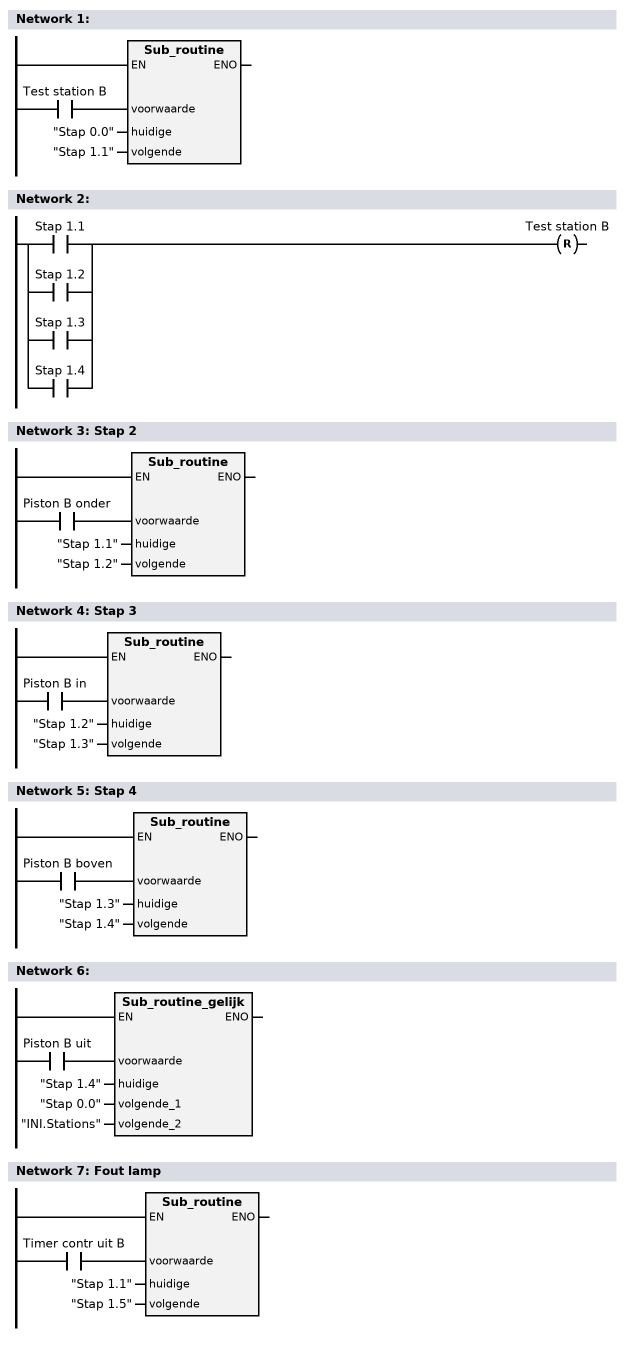
NETWORK
TITLE =
      A     "Test station B";
      =     L 0.0;
      BLD   103;
      CALL  "Sub_routine" (
           voorwaarde               := L 0.0,
           huidige                  := "Stap 0.0",
           volgende                 := "Stap 1.1");
      NOP   0;
NETWORK
TITLE =
      O     "Stap 1.1";
      O     "Stap 1.2";
      O     "Stap 1.3";
      O     "Stap 1.4";
      R     "Test station B";
NETWORK
TITLE = Stap 2
      A     "Piston B onder";
      =     L 0.0;
      BLD   103;
      CALL  "Sub_routine" (
           voorwaarde               := L 0.0,
           huidige                  := "Stap 1.1",
           volgende                 := "Stap 1.2");
      NOP   0;
NETWORK
TITLE = Stap 3
      A     "Piston B in";
      =     L 0.0;
      BLD   103;
      CALL  "Sub_routine" (
           voorwaarde               := L 0.0,
           huidige                  := "Stap 1.2",
           volgende                 := "Stap 1.3");
      NOP   0;
NETWORK
TITLE = Stap 4
      A     "Piston B boven";
      =     L 0.0;
      BLD   103;
      CALL  "Sub_routine" (
           voorwaarde               := L 0.0,
           huidige                  := "Stap 1.3",
           volgende                 := "Stap 1.4");
      NOP   0;
NETWORK
TITLE =
      A     "Piston B uit";
      =     L 0.0;
      BLD   103;
      CALL  "Sub_routine_gelijk" (
           voorwaarde               := L 0.0,
           huidige                  := "Stap 1.4",
           volgende_1               := "Stap 0.0",
           volgende_2               := "INI.Stations");
      NOP   0;
NETWORK
TITLE = Fout lamp
      A     "Timer contr uit B";
      =     L 0.0;
      BLD   103;
      CALL  "Sub_routine" (
           voorwaarde               := L 0.0,
           huidige                  := "Stap 1.1",
           volgende                 := "Stap 1.5");
      NOP   0;
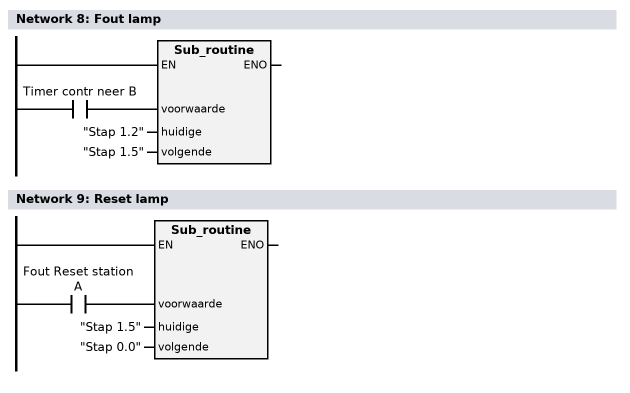
NETWORK
TITLE = Fout lamp
      A     "Timer contr neer B";
      =     L 0.0;
      BLD   103;
      CALL  "Sub_routine" (
           voorwaarde               := L 0.0,
           huidige                  := "Stap 1.2",
           volgende                 := "Stap 1.5");
      NOP   0;
NETWORK
TITLE = Reset lamp
      A     "Fout Reset station A";
      =     L 0.0;
      BLD   103;
      CALL  "Sub_routine" (
           voorwaarde               := L 0.0,
           huidige                  := "Stap 1.5",
           volgende                 := "Stap 0.0");
      NOP   0;
END_FUNCTION

FUNCTION "Simulatie_Run" : VOID	// FC 5
VERSION : 0.1
BEGIN
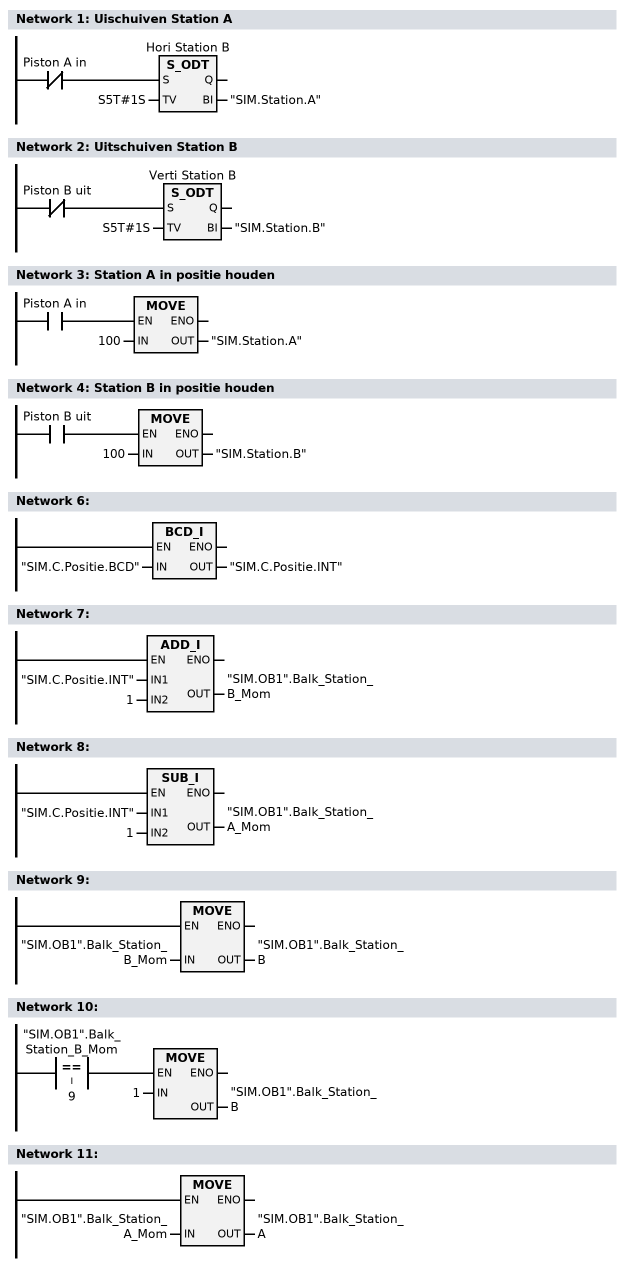
NETWORK
TITLE = Uischuiven Station A
      AN    "Piston A in";
      L     S5T#1S;
      SD    "Hori Station B";
      NOP   0;
      L     "Hori Station B";
      T     "SIM.Station.A";
      NOP   0;
      NOP   0;
NETWORK
TITLE = Uitschuiven Station B
      AN    "Piston B uit";
      L     S5T#1S;
      SD    "Verti Station B";
      NOP   0;
      L     "Verti Station B";
      T     "SIM.Station.B";
      NOP   0;
      NOP   0;
NETWORK
TITLE = Station A in positie houden
      A     "Piston A in";
      JNB   _001;
      L     100;
      T     "SIM.Station.A";
_001: NOP   0;
NETWORK
TITLE = Station B in positie houden
      A     "Piston B uit";
      JNB   _002;
      L     100;
      T     "SIM.Station.B";
_002: NOP   0;
NETWORK
TITLE = Balk voor de sensoren
      A     "Proxi Pos 2";
      AN    "Proxi Pos 1";
      FP    M 40.0;
      CU    "SIM.Positie.Staven";
      BLD   101;
      A     "Proxi Pos 1";
      FP    M 40.1;
      L     C#1;
      S     "SIM.Positie.Staven";
      NOP   0;
      NOP   0;
      LC    "SIM.Positie.Staven";
      T     "SIM.C.Positie.BCD";
      NOP   0;
NETWORK
TITLE =
      L     "SIM.C.Positie.BCD";
      BTI;
      T     "SIM.C.Positie.INT";
      NOP   0;
NETWORK
TITLE =
      L     "SIM.C.Positie.INT";
      L     1;
      +I;
      T     "SIM.OB1".Balk_Station_B_Mom;
      NOP   0;
NETWORK
TITLE =
      L     "SIM.C.Positie.INT";
      L     1;
      -I;
      T     "SIM.OB1".Balk_Station_A_Mom;
      NOP   0;
NETWORK
TITLE =
      L     "SIM.OB1".Balk_Station_B_Mom;
      T     "SIM.OB1".Balk_Station_B;
      NOP   0;
NETWORK
TITLE =
      A(;
      L     "SIM.OB1".Balk_Station_B_Mom;
      L     9;
      ==I;
      );
      JNB   _003;
      L     1;
      T     "SIM.OB1".Balk_Station_B;
_003: NOP   0;
NETWORK
TITLE =
      L     "SIM.OB1".Balk_Station_A_Mom;
      T     "SIM.OB1".Balk_Station_A;
      NOP   0;
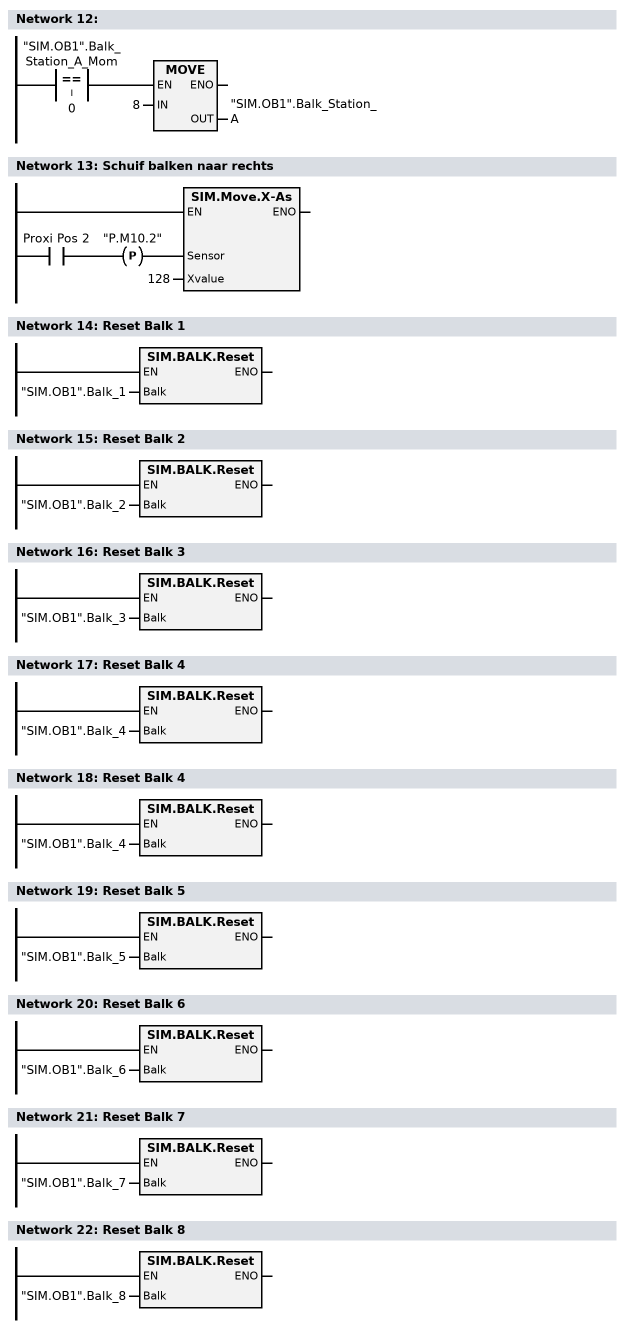
NETWORK
TITLE =
      A(;
      L     "SIM.OB1".Balk_Station_A_Mom;
      L     0;
      ==I;
      );
      JNB   _004;
      L     8;
      T     "SIM.OB1".Balk_Station_A;
_004: NOP   0;
NETWORK
TITLE = Schuif balken naar rechts
      A     "Proxi Pos 2";
      FP    "P.M10.2";
      =     L 0.0;
      BLD   103;
      CALL  "SIM.Move.X-As" (
           Sensor                   := L 0.0,
           Xvalue                   := 128);
      NOP   0;
NETWORK
TITLE = Reset Balk 1
      CALL  "SIM.BALK.Reset" (
           Balk                     := "SIM.OB1".Balk_1);
      NOP   0;
NETWORK
TITLE = Reset Balk 2
      CALL  "SIM.BALK.Reset" (
           Balk                     := "SIM.OB1".Balk_2);
      NOP   0;
NETWORK
TITLE = Reset Balk 3
      CALL  "SIM.BALK.Reset" (
           Balk                     := "SIM.OB1".Balk_3);
      NOP   0;
NETWORK
TITLE = Reset Balk 4
      CALL  "SIM.BALK.Reset" (
           Balk                     := "SIM.OB1".Balk_4);
      NOP   0;
NETWORK
TITLE = Reset Balk 4
      CALL  "SIM.BALK.Reset" (
           Balk                     := "SIM.OB1".Balk_4);
      NOP   0;
NETWORK
TITLE = Reset Balk 5
      CALL  "SIM.BALK.Reset" (
           Balk                     := "SIM.OB1".Balk_5);
      NOP   0;
NETWORK
TITLE = Reset Balk 6
      CALL  "SIM.BALK.Reset" (
           Balk                     := "SIM.OB1".Balk_6);
      NOP   0;
NETWORK
TITLE = Reset Balk 7
      CALL  "SIM.BALK.Reset" (
           Balk                     := "SIM.OB1".Balk_7);
      NOP   0;
NETWORK
TITLE = Reset Balk 8
      CALL  "SIM.BALK.Reset" (
           Balk                     := "SIM.OB1".Balk_8);
      NOP   0;
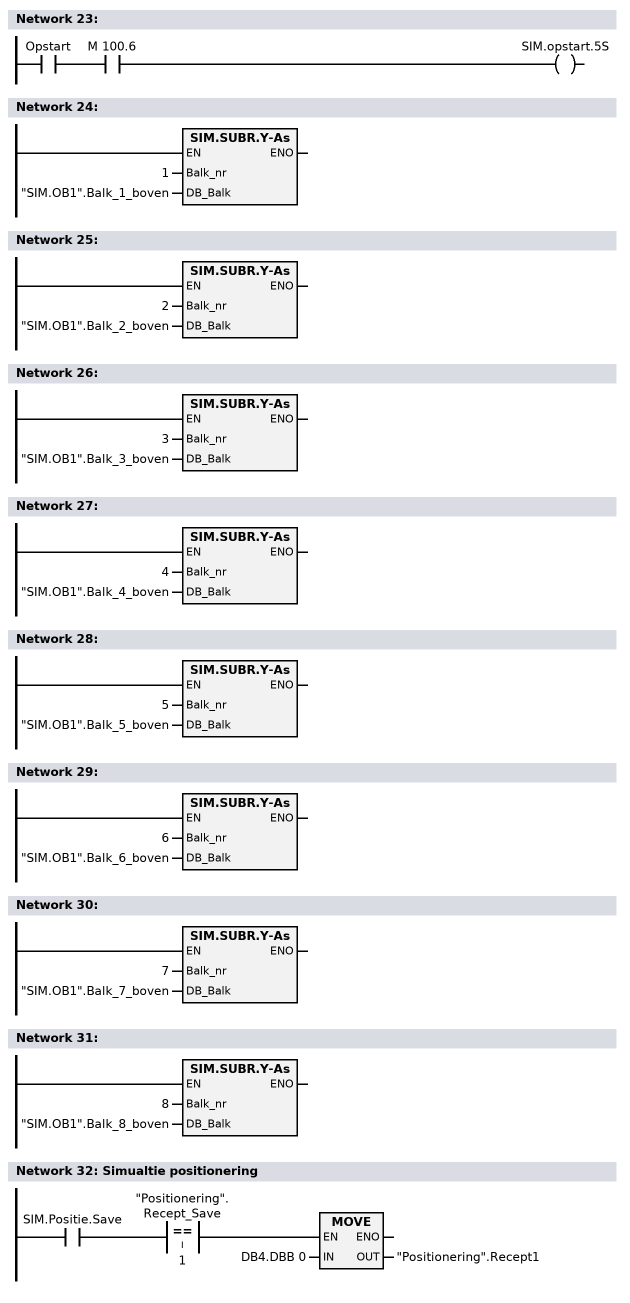
NETWORK
TITLE =
      A     "Opstart";
      A     M 100.6;
      =     "SIM.opstart.5S";
NETWORK
TITLE =
      CALL  "SIM.SUBR.Y-As" (
           Balk_nr                  := 1,
           DB_Balk                  := "SIM.OB1".Balk_1_boven);
      NOP   0;
NETWORK
TITLE =
      CALL  "SIM.SUBR.Y-As" (
           Balk_nr                  := 2,
           DB_Balk                  := "SIM.OB1".Balk_2_boven);
      NOP   0;
NETWORK
TITLE =
      CALL  "SIM.SUBR.Y-As" (
           Balk_nr                  := 3,
           DB_Balk                  := "SIM.OB1".Balk_3_boven);
      NOP   0;
NETWORK
TITLE =
      CALL  "SIM.SUBR.Y-As" (
           Balk_nr                  := 4,
           DB_Balk                  := "SIM.OB1".Balk_4_boven);
      NOP   0;
NETWORK
TITLE =
      CALL  "SIM.SUBR.Y-As" (
           Balk_nr                  := 5,
           DB_Balk                  := "SIM.OB1".Balk_5_boven);
      NOP   0;
NETWORK
TITLE =
      CALL  "SIM.SUBR.Y-As" (
           Balk_nr                  := 6,
           DB_Balk                  := "SIM.OB1".Balk_6_boven);
      NOP   0;
NETWORK
TITLE =
      CALL  "SIM.SUBR.Y-As" (
           Balk_nr                  := 7,
           DB_Balk                  := "SIM.OB1".Balk_7_boven);
      NOP   0;
NETWORK
TITLE =
      CALL  "SIM.SUBR.Y-As" (
           Balk_nr                  := 8,
           DB_Balk                  := "SIM.OB1".Balk_8_boven);
      NOP   0;
NETWORK
TITLE = Simualtie positionering
      A     "SIM.Positie.Save";
      A(;
      L     "Positionering".Recept_Save;
      L     1;
      ==I;
      );
      JNB   _005;
      L     DB4.DBB 0;
      T     "Positionering".Recept1;
_005: NOP   0;
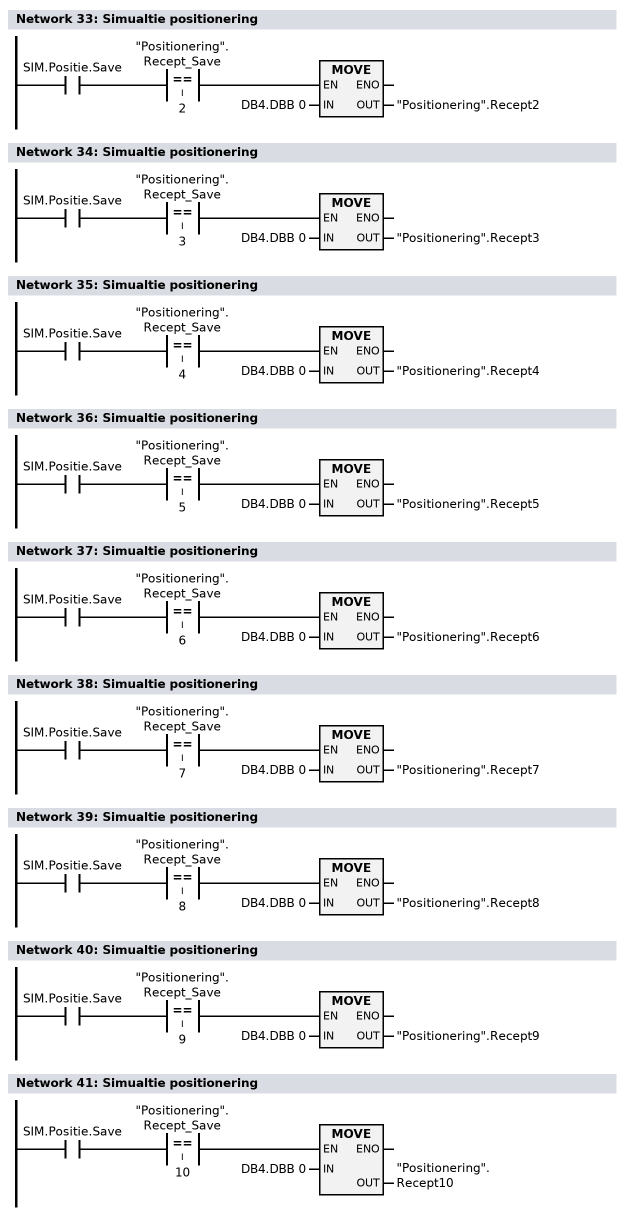
NETWORK
TITLE = Simualtie positionering
      A     "SIM.Positie.Save";
      A(;
      L     "Positionering".Recept_Save;
      L     2;
      ==I;
      );
      JNB   _006;
      L     DB4.DBB 0;
      T     "Positionering".Recept2;
_006: NOP   0;
NETWORK
TITLE = Simualtie positionering
      A     "SIM.Positie.Save";
      A(;
      L     "Positionering".Recept_Save;
      L     3;
      ==I;
      );
      JNB   _007;
      L     DB4.DBB 0;
      T     "Positionering".Recept3;
_007: NOP   0;
NETWORK
TITLE = Simualtie positionering
      A     "SIM.Positie.Save";
      A(;
      L     "Positionering".Recept_Save;
      L     4;
      ==I;
      );
      JNB   _008;
      L     DB4.DBB 0;
      T     "Positionering".Recept4;
_008: NOP   0;
NETWORK
TITLE = Simualtie positionering
      A     "SIM.Positie.Save";
      A(;
      L     "Positionering".Recept_Save;
      L     5;
      ==I;
      );
      JNB   _009;
      L     DB4.DBB 0;
      T     "Positionering".Recept5;
_009: NOP   0;
NETWORK
TITLE = Simualtie positionering
      A     "SIM.Positie.Save";
      A(;
      L     "Positionering".Recept_Save;
      L     6;
      ==I;
      );
      JNB   _00a;
      L     DB4.DBB 0;
      T     "Positionering".Recept6;
_00a: NOP   0;
NETWORK
TITLE = Simualtie positionering
      A     "SIM.Positie.Save";
      A(;
      L     "Positionering".Recept_Save;
      L     7;
      ==I;
      );
      JNB   _00b;
      L     DB4.DBB 0;
      T     "Positionering".Recept7;
_00b: NOP   0;
NETWORK
TITLE = Simualtie positionering
      A     "SIM.Positie.Save";
      A(;
      L     "Positionering".Recept_Save;
      L     8;
      ==I;
      );
      JNB   _00c;
      L     DB4.DBB 0;
      T     "Positionering".Recept8;
_00c: NOP   0;
NETWORK
TITLE = Simualtie positionering
      A     "SIM.Positie.Save";
      A(;
      L     "Positionering".Recept_Save;
      L     9;
      ==I;
      );
      JNB   _00d;
      L     DB4.DBB 0;
      T     "Positionering".Recept9;
_00d: NOP   0;
NETWORK
TITLE = Simualtie positionering
      A     "SIM.Positie.Save";
      A(;
      L     "Positionering".Recept_Save;
      L     10;
      ==I;
      );
      JNB   _00e;
      L     DB4.DBB 0;
      T     "Positionering".Recept10;
_00e: NOP   0;
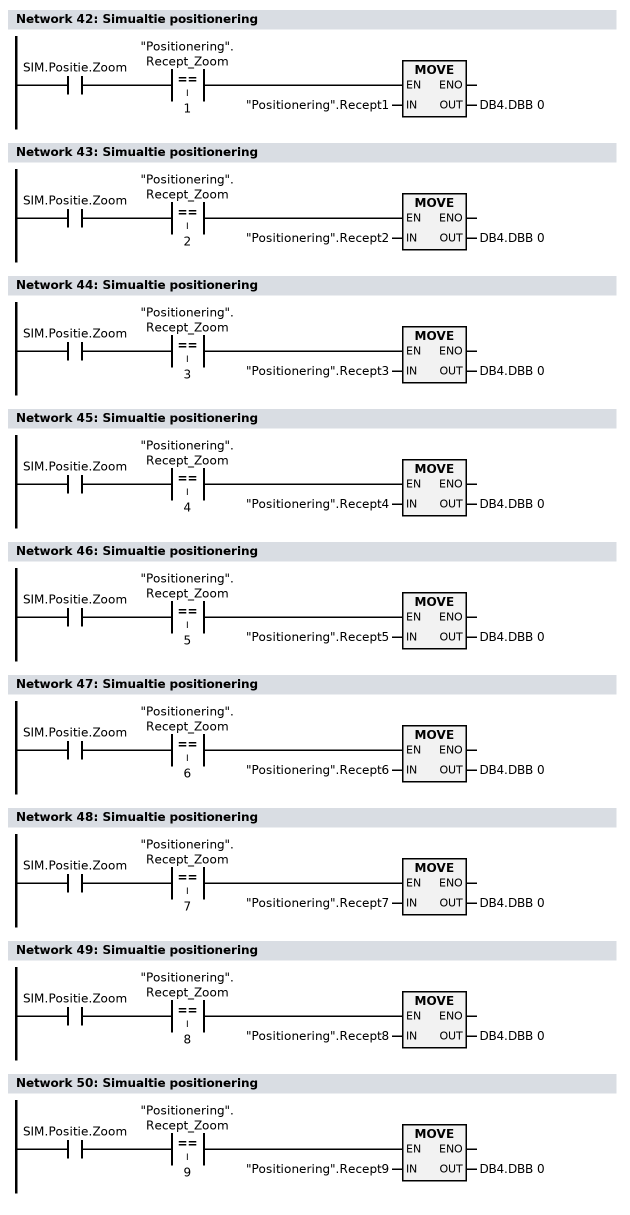
NETWORK
TITLE = Simualtie positionering
      A     "SIM.Positie.Zoom";
      A(;
      L     "Positionering".Recept_Zoom;
      L     1;
      ==I;
      );
      JNB   _00f;
      L     "Positionering".Recept1;
      T     DB4.DBB 0;
_00f: NOP   0;
NETWORK
TITLE = Simualtie positionering
      A     "SIM.Positie.Zoom";
      A(;
      L     "Positionering".Recept_Zoom;
      L     2;
      ==I;
      );
      JNB   _010;
      L     "Positionering".Recept2;
      T     DB4.DBB 0;
_010: NOP   0;
NETWORK
TITLE = Simualtie positionering
      A     "SIM.Positie.Zoom";
      A(;
      L     "Positionering".Recept_Zoom;
      L     3;
      ==I;
      );
      JNB   _011;
      L     "Positionering".Recept3;
      T     DB4.DBB 0;
_011: NOP   0;
NETWORK
TITLE = Simualtie positionering
      A     "SIM.Positie.Zoom";
      A(;
      L     "Positionering".Recept_Zoom;
      L     4;
      ==I;
      );
      JNB   _012;
      L     "Positionering".Recept4;
      T     DB4.DBB 0;
_012: NOP   0;
NETWORK
TITLE = Simualtie positionering
      A     "SIM.Positie.Zoom";
      A(;
      L     "Positionering".Recept_Zoom;
      L     5;
      ==I;
      );
      JNB   _013;
      L     "Positionering".Recept5;
      T     DB4.DBB 0;
_013: NOP   0;
NETWORK
TITLE = Simualtie positionering
      A     "SIM.Positie.Zoom";
      A(;
      L     "Positionering".Recept_Zoom;
      L     6;
      ==I;
      );
      JNB   _014;
      L     "Positionering".Recept6;
      T     DB4.DBB 0;
_014: NOP   0;
NETWORK
TITLE = Simualtie positionering
      A     "SIM.Positie.Zoom";
      A(;
      L     "Positionering".Recept_Zoom;
      L     7;
      ==I;
      );
      JNB   _015;
      L     "Positionering".Recept7;
      T     DB4.DBB 0;
_015: NOP   0;
NETWORK
TITLE = Simualtie positionering
      A     "SIM.Positie.Zoom";
      A(;
      L     "Positionering".Recept_Zoom;
      L     8;
      ==I;
      );
      JNB   _016;
      L     "Positionering".Recept8;
      T     DB4.DBB 0;
_016: NOP   0;
NETWORK
TITLE = Simualtie positionering
      A     "SIM.Positie.Zoom";
      A(;
      L     "Positionering".Recept_Zoom;
      L     9;
      ==I;
      );
      JNB   _017;
      L     "Positionering".Recept9;
      T     DB4.DBB 0;
_017: NOP   0;
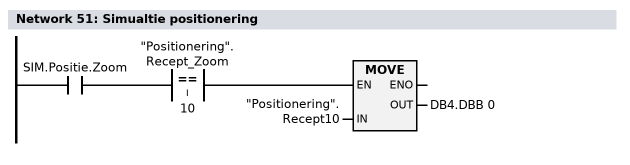
NETWORK
TITLE = Simualtie positionering
      A     "SIM.Positie.Zoom";
      A(;
      L     "Positionering".Recept_Zoom;
      L     10;
      ==I;
      );
      JNB   _018;
      L     "Positionering".Recept10;
      T     DB4.DBB 0;
_018: NOP   0;
END_FUNCTION

FUNCTION "Opstart_FC" : VOID	// FC 6
VERSION : 0.1
BEGIN
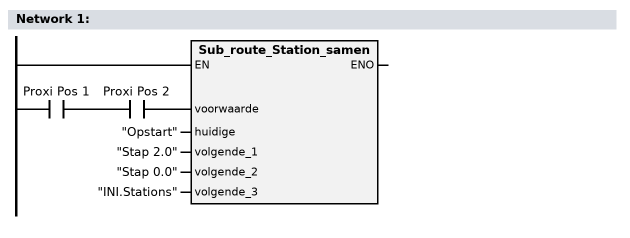
NETWORK
TITLE =
      A     "Proxi Pos 1";
      A     "Proxi Pos 2";
      =     L 0.0;
      BLD   103;
      CALL  "Sub_route_Station_samen" (
           voorwaarde               := L 0.0,
           huidige                  := "Opstart",
           volgende_1               := "Stap 2.0",
           volgende_2               := "Stap 0.0",
           volgende_3               := "INI.Stations");
      NOP   0;
END_FUNCTION

FUNCTION "Grafcet_Platform" : VOID	// FC 7
VERSION : 0.1
BEGIN
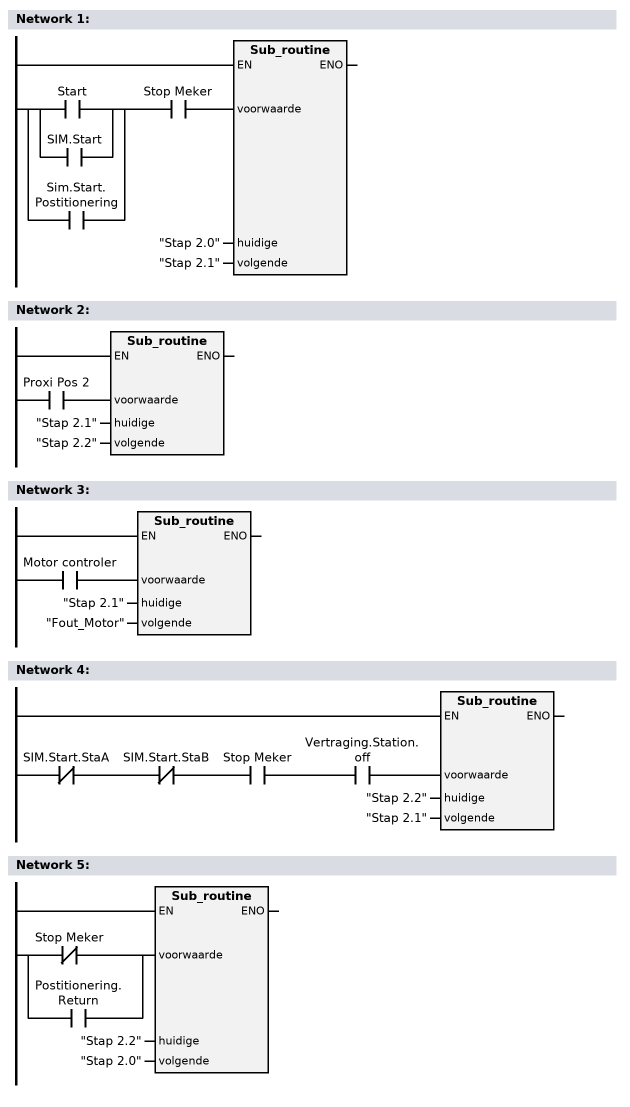
NETWORK
TITLE =
      A(;
      O     "Start";
      O     "SIM.Start";
      O     "Sim.Start.Postitionering";
      );
      A     "Stop Meker";
      =     L 0.0;
      BLD   103;
      CALL  "Sub_routine" (
           voorwaarde               := L 0.0,
           huidige                  := "Stap 2.0",
           volgende                 := "Stap 2.1");
      NOP   0;
NETWORK
TITLE =
      A     "Proxi Pos 2";
      =     L 0.0;
      BLD   103;
      CALL  "Sub_routine" (
           voorwaarde               := L 0.0,
           huidige                  := "Stap 2.1",
           volgende                 := "Stap 2.2");
      NOP   0;
NETWORK
TITLE =
      A     "Motor controler";
      =     L 0.0;
      BLD   103;
      CALL  "Sub_routine" (
           voorwaarde               := L 0.0,
           huidige                  := "Stap 2.1",
           volgende                 := "Fout_Motor");
      NOP   0;
NETWORK
TITLE =
      AN    "SIM.Start.StaA";
      AN    "SIM.Start.StaB";
      A     "Stop Meker";
      A     "Vertraging.Station.off";
      =     L 0.0;
      BLD   103;
      CALL  "Sub_routine" (
           voorwaarde               := L 0.0,
           huidige                  := "Stap 2.2",
           volgende                 := "Stap 2.1");
      NOP   0;
NETWORK
TITLE =
      A(;
      ON    "Stop Meker";
      O     "Postitionering.Return";
      );
      =     L 0.0;
      BLD   103;
      CALL  "Sub_routine" (
           voorwaarde               := L 0.0,
           huidige                  := "Stap 2.2",
           volgende                 := "Stap 2.0");
      NOP   0;
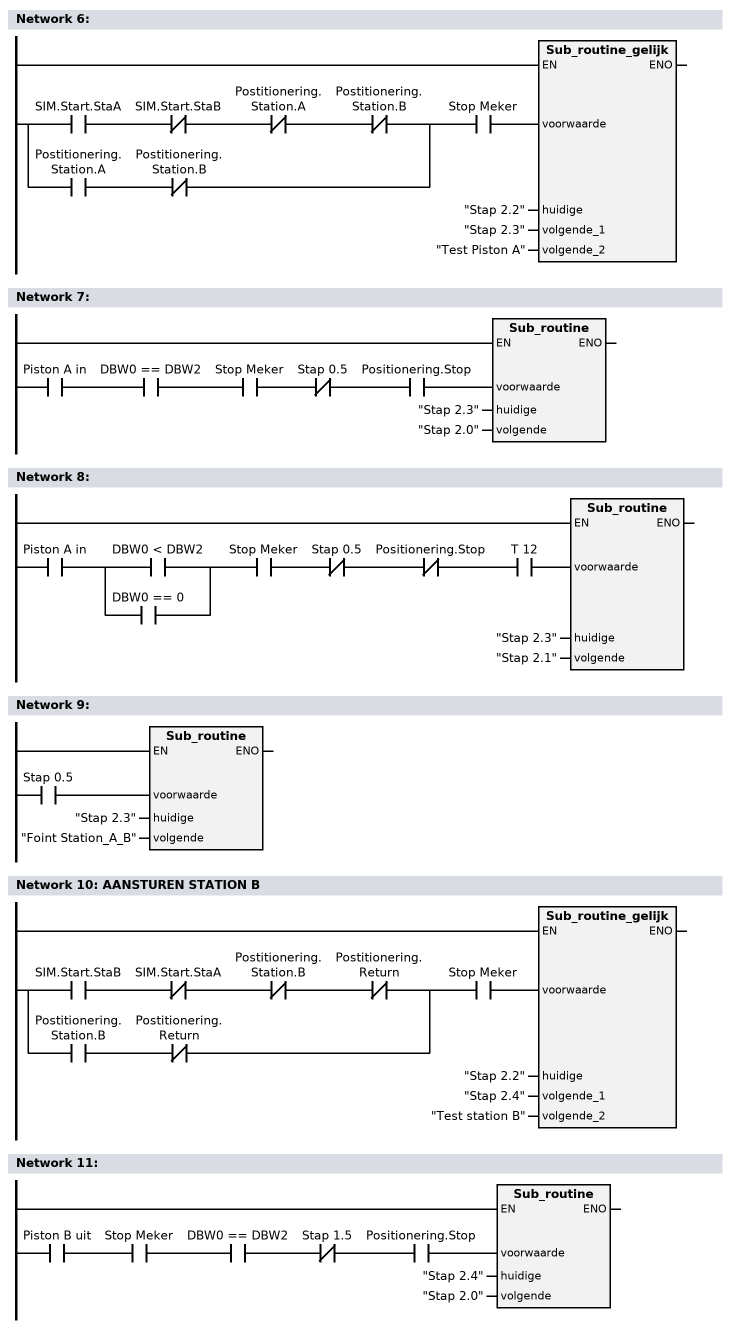
NETWORK
TITLE =
      A(;
      A     "SIM.Start.StaA";
      AN    "SIM.Start.StaB";
      AN    "Postitionering.Station.A";
      AN    "Postitionering.Station.B";
      O;
      A     "Postitionering.Station.A";
      AN    "Postitionering.Station.B";
      );
      A     "Stop Meker";
      =     L 0.0;
      BLD   103;
      CALL  "Sub_routine_gelijk" (
           voorwaarde               := L 0.0,
           huidige                  := "Stap 2.2",
           volgende_1               := "Stap 2.3",
           volgende_2               := "Test Piston A");
      NOP   0;
NETWORK
TITLE =
      A     "Piston A in";
      A     "DBW0 == DBW2";
      A     "Stop Meker";
      AN    "Stap 0.5";
      A     "Positionering.Stop";
      =     L 0.0;
      BLD   103;
      CALL  "Sub_routine" (
           voorwaarde               := L 0.0,
           huidige                  := "Stap 2.3",
           volgende                 := "Stap 2.0");
      NOP   0;
NETWORK
TITLE =
      A     "Piston A in";
      A(;
      O     "DBW0 < DBW2";
      O     "DBW0 == 0";
      );
      A     "Stop Meker";
      AN    "Stap 0.5";
      AN    "Positionering.Stop";
      A     T 12;
      =     L 0.0;
      BLD   103;
      CALL  "Sub_routine" (
           voorwaarde               := L 0.0,
           huidige                  := "Stap 2.3",
           volgende                 := "Stap 2.1");
      NOP   0;
NETWORK
TITLE =
      A     "Stap 0.5";
      =     L 0.0;
      BLD   103;
      CALL  "Sub_routine" (
           voorwaarde               := L 0.0,
           huidige                  := "Stap 2.3",
           volgende                 := "Foint Station_A_B");
      NOP   0;
NETWORK
TITLE = AANSTUREN STATION B
      A(;
      A     "SIM.Start.StaB";
      AN    "SIM.Start.StaA";
      AN    "Postitionering.Station.B";
      AN    "Postitionering.Return";
      O;
      A     "Postitionering.Station.B";
      AN    "Postitionering.Return";
      );
      A     "Stop Meker";
      =     L 0.0;
      BLD   103;
      CALL  "Sub_routine_gelijk" (
           voorwaarde               := L 0.0,
           huidige                  := "Stap 2.2",
           volgende_1               := "Stap 2.4",
           volgende_2               := "Test station B");
      NOP   0;
NETWORK
TITLE =
      A     "Piston B uit";
      A     "Stop Meker";
      A     "DBW0 == DBW2";
      AN    "Stap 1.5";
      A     "Positionering.Stop";
      =     L 0.0;
      BLD   103;
      CALL  "Sub_routine" (
           voorwaarde               := L 0.0,
           huidige                  := "Stap 2.4",
           volgende                 := "Stap 2.0");
      NOP   0;
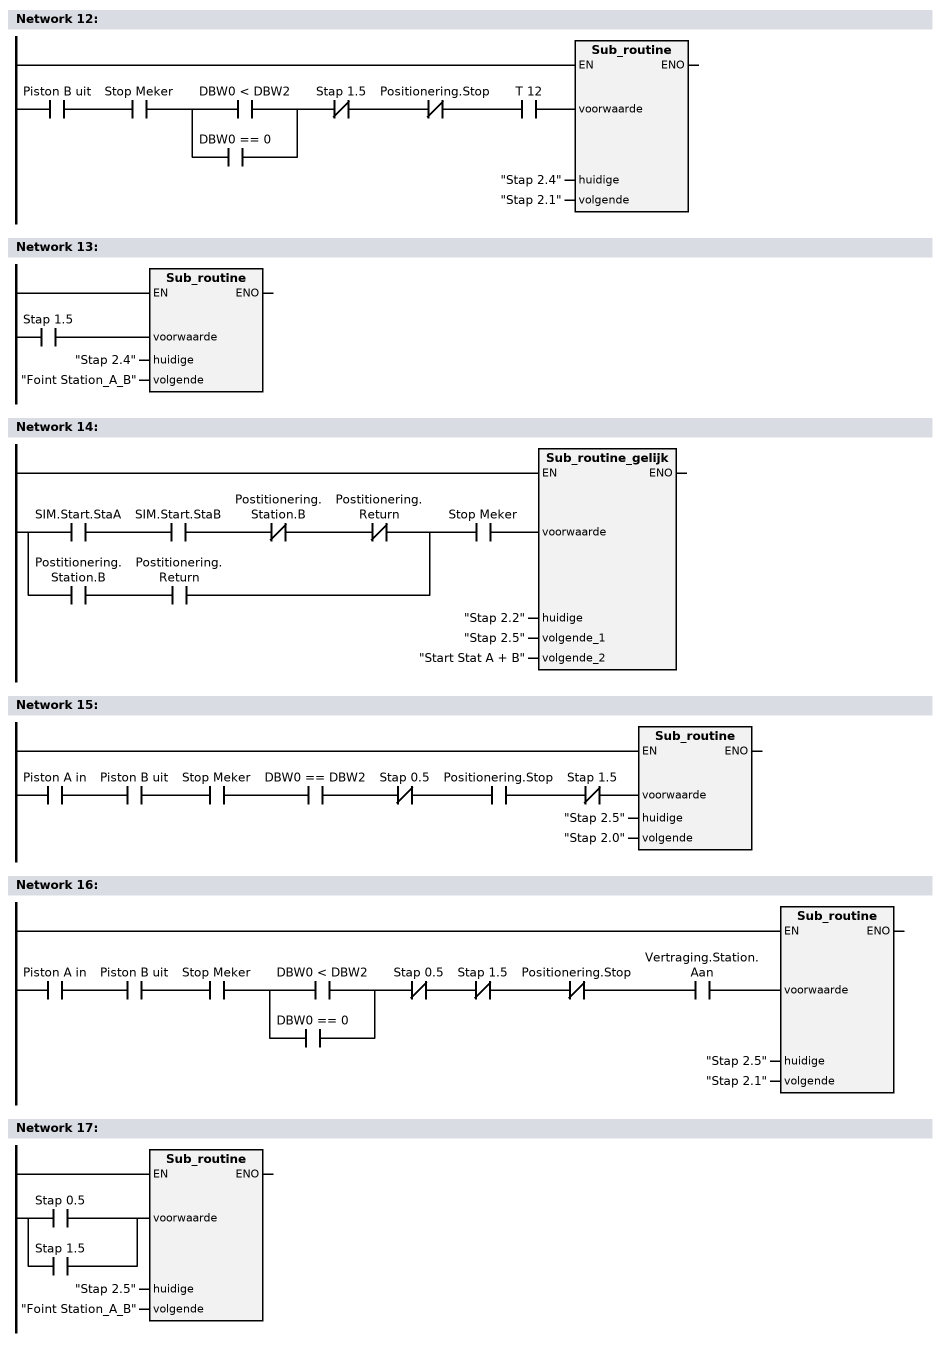
NETWORK
TITLE =
      A     "Piston B uit";
      A     "Stop Meker";
      A(;
      O     "DBW0 < DBW2";
      O     "DBW0 == 0";
      );
      AN    "Stap 1.5";
      AN    "Positionering.Stop";
      A     T 12;
      =     L 0.0;
      BLD   103;
      CALL  "Sub_routine" (
           voorwaarde               := L 0.0,
           huidige                  := "Stap 2.4",
           volgende                 := "Stap 2.1");
      NOP   0;
NETWORK
TITLE =
      A     "Stap 1.5";
      =     L 0.0;
      BLD   103;
      CALL  "Sub_routine" (
           voorwaarde               := L 0.0,
           huidige                  := "Stap 2.4",
           volgende                 := "Foint Station_A_B");
      NOP   0;
NETWORK
TITLE =
      A(;
      A     "SIM.Start.StaA";
      A     "SIM.Start.StaB";
      AN    "Postitionering.Station.B";
      AN    "Postitionering.Return";
      O;
      A     "Postitionering.Station.B";
      A     "Postitionering.Return";
      );
      A     "Stop Meker";
      =     L 0.0;
      BLD   103;
      CALL  "Sub_routine_gelijk" (
           voorwaarde               := L 0.0,
           huidige                  := "Stap 2.2",
           volgende_1               := "Stap 2.5",
           volgende_2               := "Start Stat A + B");
      NOP   0;
NETWORK
TITLE =
      A     "Piston A in";
      A     "Piston B uit";
      A     "Stop Meker";
      A     "DBW0 == DBW2";
      AN    "Stap 0.5";
      A     "Positionering.Stop";
      AN    "Stap 1.5";
      =     L 0.0;
      BLD   103;
      CALL  "Sub_routine" (
           voorwaarde               := L 0.0,
           huidige                  := "Stap 2.5",
           volgende                 := "Stap 2.0");
      NOP   0;
NETWORK
TITLE =
      A     "Piston A in";
      A     "Piston B uit";
      A     "Stop Meker";
      A(;
      O     "DBW0 < DBW2";
      O     "DBW0 == 0";
      );
      AN    "Stap 0.5";
      AN    "Stap 1.5";
      AN    "Positionering.Stop";
      A     "Vertraging.Station.Aan";
      =     L 0.0;
      BLD   103;
      CALL  "Sub_routine" (
           voorwaarde               := L 0.0,
           huidige                  := "Stap 2.5",
           volgende                 := "Stap 2.1");
      NOP   0;
NETWORK
TITLE =
      A(;
      O     "Stap 0.5";
      O     "Stap 1.5";
      );
      =     L 0.0;
      BLD   103;
      CALL  "Sub_routine" (
           voorwaarde               := L 0.0,
           huidige                  := "Stap 2.5",
           volgende                 := "Foint Station_A_B");
      NOP   0;
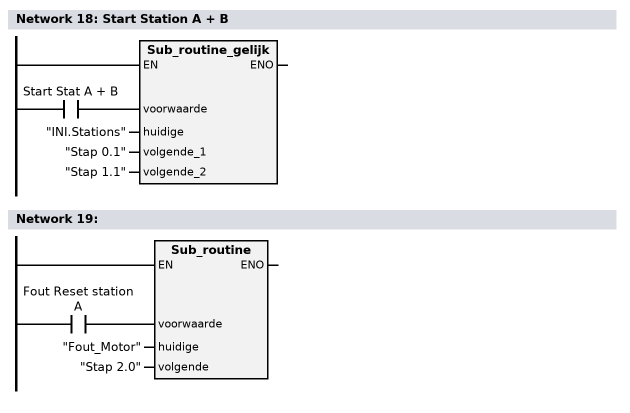
NETWORK
TITLE = Start Station A + B
      A     "Start Stat A + B";
      =     L 0.0;
      BLD   103;
      CALL  "Sub_routine_gelijk" (
           voorwaarde               := L 0.0,
           huidige                  := "INI.Stations",
           volgende_1               := "Stap 0.1",
           volgende_2               := "Stap 1.1");
      NOP   0;
NETWORK
TITLE =
      A     "Fout Reset station A";
      =     L 0.0;
      BLD   103;
      CALL  "Sub_routine" (
           voorwaarde               := L 0.0,
           huidige                  := "Fout_Motor",
           volgende                 := "Stap 2.0");
      NOP   0;
END_FUNCTION

FUNCTION "Ingang -> Merker" : VOID	// FC 8
VERSION : 0.1
BEGIN
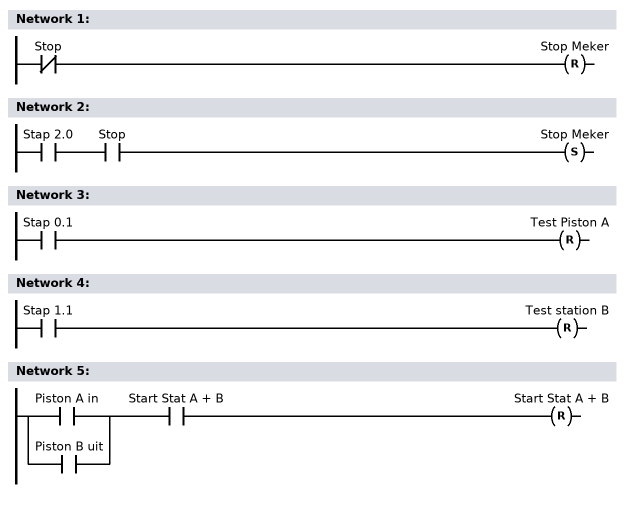
NETWORK
TITLE =
      AN    "Stop";
      R     "Stop Meker";
NETWORK
TITLE =
      A     "Stap 2.0";
      A     "Stop";
      S     "Stop Meker";
NETWORK
TITLE =
      A     "Stap 0.1";
      R     "Test Piston A";
NETWORK
TITLE =
      A     "Stap 1.1";
      R     "Test station B";
NETWORK
TITLE =
      A(;
      O     "Piston A in";
      O     "Piston B uit";
      );
      A     "Start Stat A + B";
      R     "Start Stat A + B";
END_FUNCTION

FUNCTION "DB_Function" : VOID	// FC 9
VERSION : 0.1
BEGIN
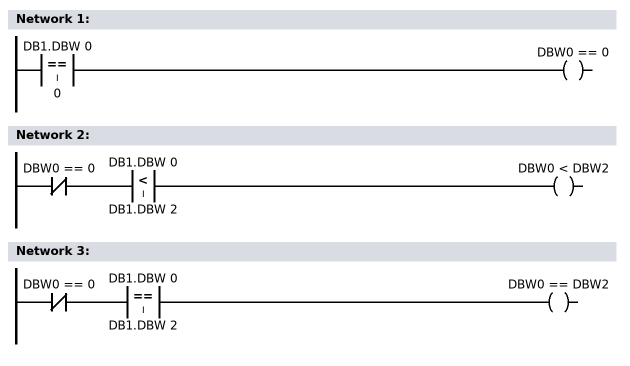
NETWORK
TITLE =
      L     DB1.DBW 0;
      L     0;
      ==I;
      =     "DBW0 == 0";
NETWORK
TITLE =
      AN    "DBW0 == 0";
      A(;
      L     DB1.DBW 0;
      L     DB1.DBW 2;
      <I;
      );
      =     "DBW0 < DBW2";
NETWORK
TITLE =
      AN    "DBW0 == 0";
      A(;
      L     DB1.DBW 0;
      L     DB1.DBW 2;
      ==I;
      );
      =     "DBW0 == DBW2";
END_FUNCTION

FUNCTION "SIM.OB100" : VOID	// FC 10
VERSION : 0.1
BEGIN
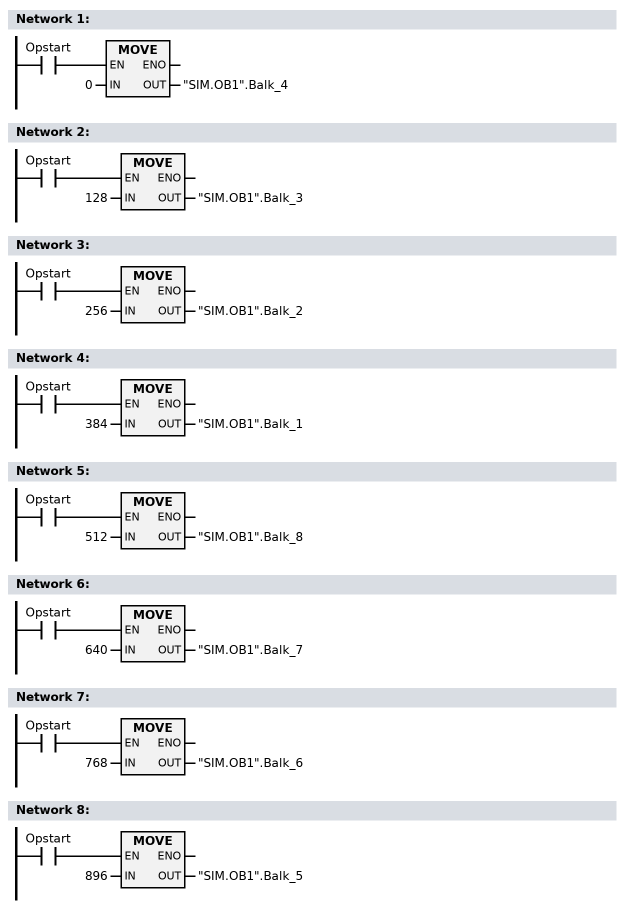
NETWORK
TITLE =
      A     "Opstart";
      JNB   _001;
      L     0;
      T     "SIM.OB1".Balk_4;
_001: NOP   0;
NETWORK
TITLE =
      A     "Opstart";
      JNB   _002;
      L     128;
      T     "SIM.OB1".Balk_3;
_002: NOP   0;
NETWORK
TITLE =
      A     "Opstart";
      JNB   _003;
      L     256;
      T     "SIM.OB1".Balk_2;
_003: NOP   0;
NETWORK
TITLE =
      A     "Opstart";
      JNB   _004;
      L     384;
      T     "SIM.OB1".Balk_1;
_004: NOP   0;
NETWORK
TITLE =
      A     "Opstart";
      JNB   _005;
      L     512;
      T     "SIM.OB1".Balk_8;
_005: NOP   0;
NETWORK
TITLE =
      A     "Opstart";
      JNB   _006;
      L     640;
      T     "SIM.OB1".Balk_7;
_006: NOP   0;
NETWORK
TITLE =
      A     "Opstart";
      JNB   _007;
      L     768;
      T     "SIM.OB1".Balk_6;
_007: NOP   0;
NETWORK
TITLE =
      A     "Opstart";
      JNB   _008;
      L     896;
      T     "SIM.OB1".Balk_5;
_008: NOP   0;
END_FUNCTION

FUNCTION "SIM.user" : VOID	// FC 11
VERSION : 0.1
BEGIN
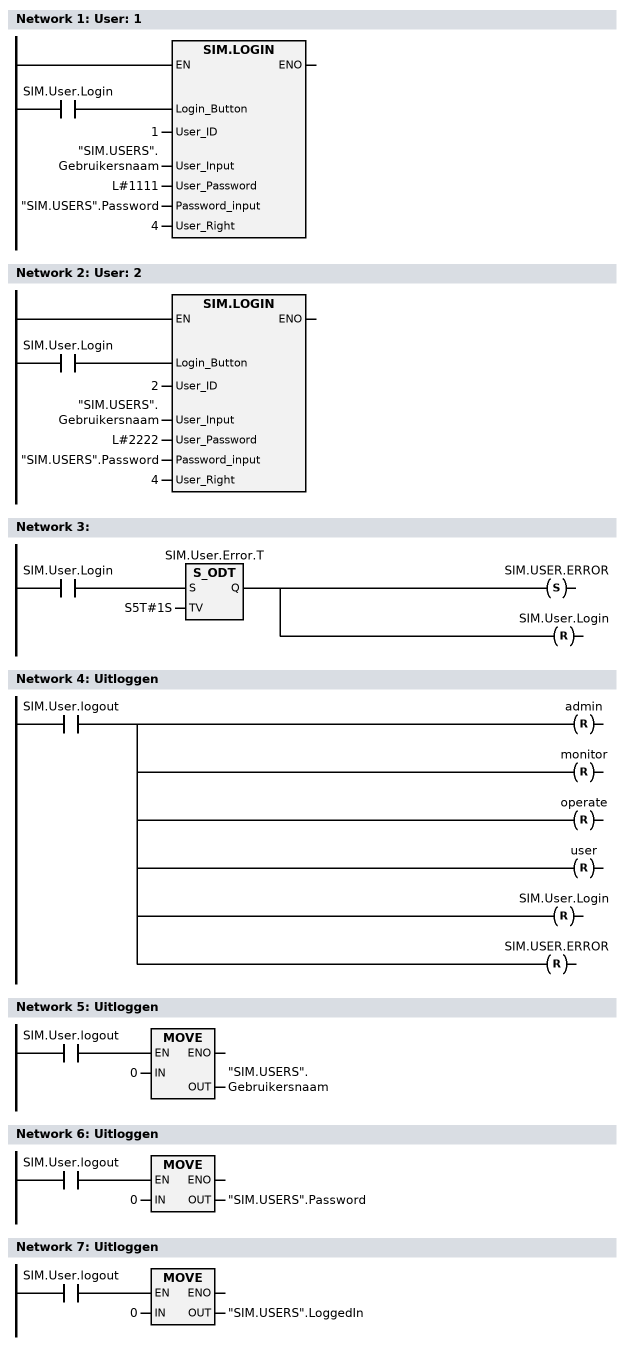
NETWORK
TITLE = User: 1
      A     "SIM.User.Login";
      =     L 0.0;
      BLD   103;
      CALL  "SIM.LOGIN" (
           Login_Button             := L 0.0,
           User_ID                  := 1,
           User_Input               := "SIM.USERS".Gebruikersnaam,
           User_Password            := L#1111,
           Password_input           := "SIM.USERS".Password,
           User_Right               := 4);
      NOP   0;
NETWORK
TITLE = User: 2
      A     "SIM.User.Login";
      =     L 0.0;
      BLD   103;
      CALL  "SIM.LOGIN" (
           Login_Button             := L 0.0,
           User_ID                  := 2,
           User_Input               := "SIM.USERS".Gebruikersnaam,
           User_Password            := L#2222,
           Password_input           := "SIM.USERS".Password,
           User_Right               := 4);
      NOP   0;
NETWORK
TITLE =
      A     "SIM.User.Login";
      L     S5T#1S;
      SD    "SIM.User.Error.T";
      NOP   0;
      NOP   0;
      NOP   0;
      A     "SIM.User.Error.T";
      S     "SIM.USER.ERROR";
      R     "SIM.User.Login";
NETWORK
TITLE = Uitloggen
      A     "SIM.User.logout";
      R     "admin";
      R     "monitor";
      R     "operate";
      R     "user";
      R     "SIM.User.Login";
      R     "SIM.USER.ERROR";
NETWORK
TITLE = Uitloggen
      A     "SIM.User.logout";
      JNB   _001;
      L     0;
      T     "SIM.USERS".Gebruikersnaam;
_001: NOP   0;
NETWORK
TITLE = Uitloggen
      A     "SIM.User.logout";
      JNB   _002;
      L     0;
      T     "SIM.USERS".Password;
_002: NOP   0;
NETWORK
TITLE = Uitloggen
      A     "SIM.User.logout";
      JNB   _003;
      L     0;
      T     "SIM.USERS".LoggedIn;
_003: NOP   0;
END_FUNCTION

FUNCTION "Positionering_balken" : VOID	// FC 12
VERSION : 0.1
VAR_TEMP
  Return_StationA_Balk1 : BOOL ;
  Return_StationA_Balk2 : BOOL ;
  Return_StationA_Balk3 : BOOL ;
  Return_StationA_Balk4 : BOOL ;
  Return_StationA_Balk5 : BOOL ;
  Return_StationA_Balk6 : BOOL ;
  Return_StationA_Balk7 : BOOL ;
  Return_StationA_Balk8 : BOOL ;
  Return_StationB_Balk1 : BOOL ;
  Return_StationB_Balk2 : BOOL ;
  Return_StationB_Balk3 : BOOL ;
  Return_StationB_Balk4 : BOOL ;
  Return_StationB_Balk5 : BOOL ;
  Return_StationB_Balk6 : BOOL ;
  Return_StationB_Balk7 : BOOL ;
  Return_StationB_Balk8 : BOOL ;
  Activatie_StationA_Balk1 : BOOL ;
  Activatie_StationA_Balk2 : BOOL ;
  Activatie_StationA_Balk3 : BOOL ;
  Activatie_StationA_Balk4 : BOOL ;
  Activatie_StationA_Balk5 : BOOL ;
  Activatie_StationA_Balk6 : BOOL ;
  Activatie_StationA_Balk7 : BOOL ;
  Activatie_StationA_Balk8 : BOOL ;
  Activatie_StationB_Balk1 : BOOL ;
  Activatie_StationB_Balk2 : BOOL ;
  Activatie_StationB_Balk3 : BOOL ;
  Activatie_StationB_Balk4 : BOOL ;
  Activatie_StationB_Balk5 : BOOL ;
  Activatie_StationB_Balk6 : BOOL ;
  Activatie_StationB_Balk7 : BOOL ;
  Activatie_StationB_Balk8 : BOOL ;
  Positief : BOOL ;
  CouterValueBCD : WORD ;
  CounterValueInt : INT ;
  ResetCounter : BOOL ;
END_VAR
BEGIN
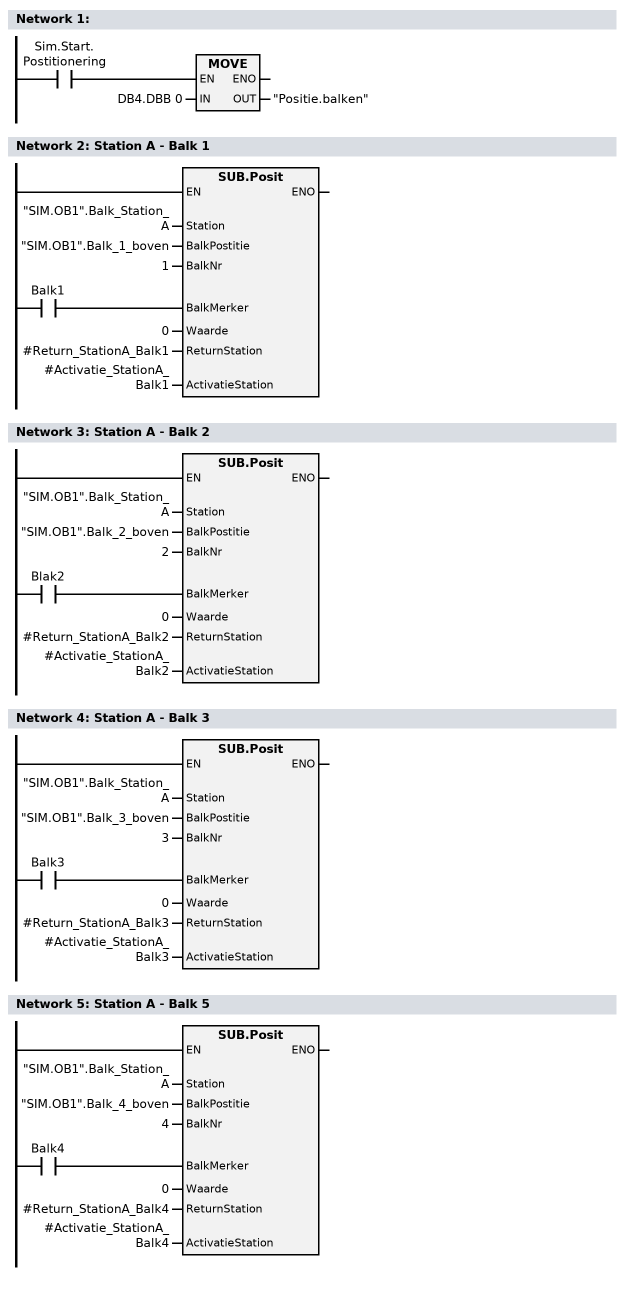
NETWORK
TITLE =
      A     "Sim.Start.Postitionering";
      JNB   _001;
      L     DB4.DBB 0;
      T     "Positie.balken";
_001: NOP   0;
NETWORK
TITLE = Station A - Balk 1
      A     "Balk1";
      =     L 11.0;
      BLD   103;
      CALL  "SUB.Posit" (
           Station                  := "SIM.OB1".Balk_Station_A,
           BalkPostitie             := "SIM.OB1".Balk_1_boven,
           BalkNr                   := 1,
           BalkMerker               := L 11.0,
           Waarde                   := 0,
           ReturnStation            := #Return_StationA_Balk1,
           ActivatieStation         := #Activatie_StationA_Balk1);
      NOP   0;
NETWORK
TITLE = Station A - Balk 2
      A     "Blak2";
      =     L 11.0;
      BLD   103;
      CALL  "SUB.Posit" (
           Station                  := "SIM.OB1".Balk_Station_A,
           BalkPostitie             := "SIM.OB1".Balk_2_boven,
           BalkNr                   := 2,
           BalkMerker               := L 11.0,
           Waarde                   := 0,
           ReturnStation            := #Return_StationA_Balk2,
           ActivatieStation         := #Activatie_StationA_Balk2);
      NOP   0;
NETWORK
TITLE = Station A - Balk 3
      A     "Balk3";
      =     L 11.0;
      BLD   103;
      CALL  "SUB.Posit" (
           Station                  := "SIM.OB1".Balk_Station_A,
           BalkPostitie             := "SIM.OB1".Balk_3_boven,
           BalkNr                   := 3,
           BalkMerker               := L 11.0,
           Waarde                   := 0,
           ReturnStation            := #Return_StationA_Balk3,
           ActivatieStation         := #Activatie_StationA_Balk3);
      NOP   0;
NETWORK
TITLE = Station A - Balk 5
      A     "Balk4";
      =     L 11.0;
      BLD   103;
      CALL  "SUB.Posit" (
           Station                  := "SIM.OB1".Balk_Station_A,
           BalkPostitie             := "SIM.OB1".Balk_4_boven,
           BalkNr                   := 4,
           BalkMerker               := L 11.0,
           Waarde                   := 0,
           ReturnStation            := #Return_StationA_Balk4,
           ActivatieStation         := #Activatie_StationA_Balk4);
      NOP   0;
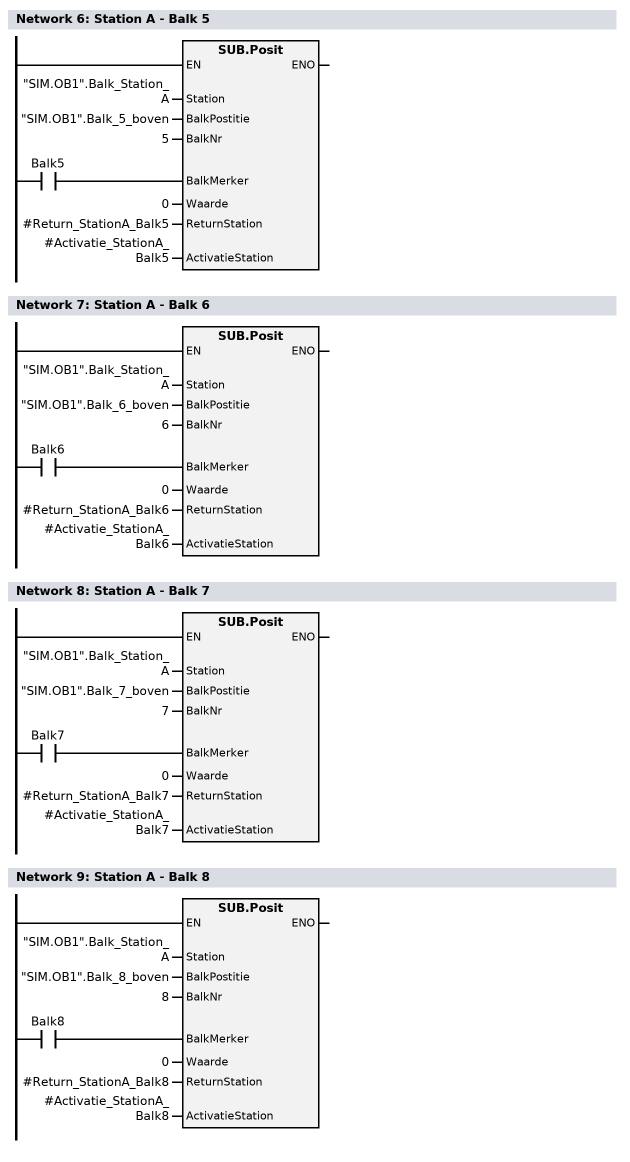
NETWORK
TITLE = Station A - Balk 5
      A     "Balk5";
      =     L 11.0;
      BLD   103;
      CALL  "SUB.Posit" (
           Station                  := "SIM.OB1".Balk_Station_A,
           BalkPostitie             := "SIM.OB1".Balk_5_boven,
           BalkNr                   := 5,
           BalkMerker               := L 11.0,
           Waarde                   := 0,
           ReturnStation            := #Return_StationA_Balk5,
           ActivatieStation         := #Activatie_StationA_Balk5);
      NOP   0;
NETWORK
TITLE = Station A - Balk 6
      A     "Balk6";
      =     L 11.0;
      BLD   103;
      CALL  "SUB.Posit" (
           Station                  := "SIM.OB1".Balk_Station_A,
           BalkPostitie             := "SIM.OB1".Balk_6_boven,
           BalkNr                   := 6,
           BalkMerker               := L 11.0,
           Waarde                   := 0,
           ReturnStation            := #Return_StationA_Balk6,
           ActivatieStation         := #Activatie_StationA_Balk6);
      NOP   0;
NETWORK
TITLE = Station A - Balk 7
      A     "Balk7";
      =     L 11.0;
      BLD   103;
      CALL  "SUB.Posit" (
           Station                  := "SIM.OB1".Balk_Station_A,
           BalkPostitie             := "SIM.OB1".Balk_7_boven,
           BalkNr                   := 7,
           BalkMerker               := L 11.0,
           Waarde                   := 0,
           ReturnStation            := #Return_StationA_Balk7,
           ActivatieStation         := #Activatie_StationA_Balk7);
      NOP   0;
NETWORK
TITLE = Station A - Balk 8
      A     "Balk8";
      =     L 11.0;
      BLD   103;
      CALL  "SUB.Posit" (
           Station                  := "SIM.OB1".Balk_Station_A,
           BalkPostitie             := "SIM.OB1".Balk_8_boven,
           BalkNr                   := 8,
           BalkMerker               := L 11.0,
           Waarde                   := 0,
           ReturnStation            := #Return_StationA_Balk8,
           ActivatieStation         := #Activatie_StationA_Balk8);
      NOP   0;
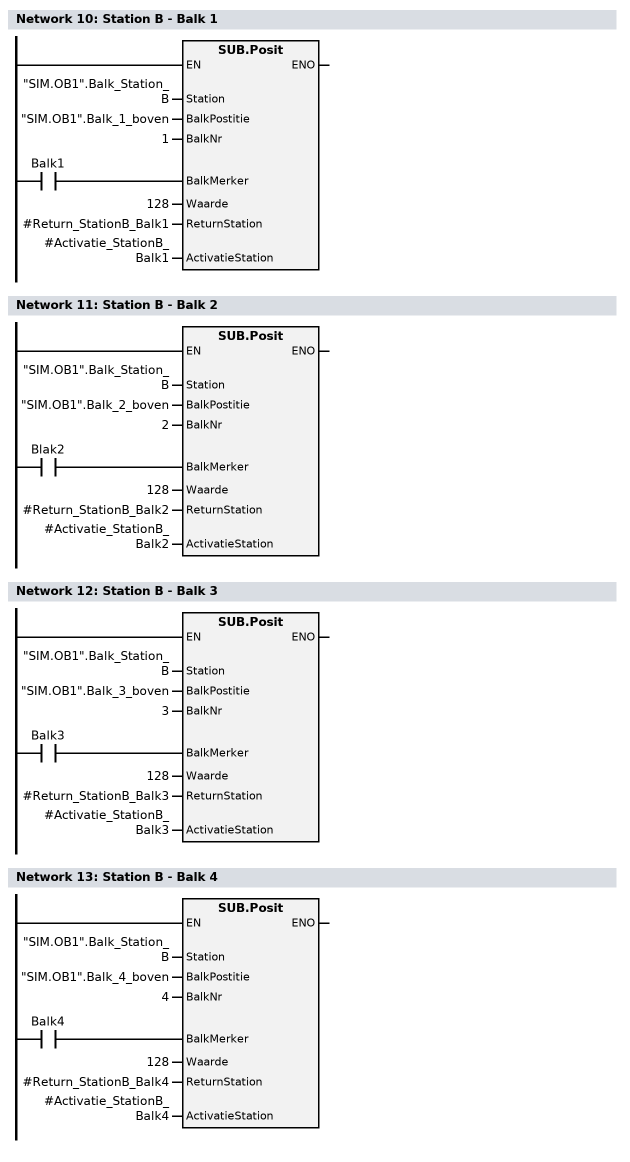
NETWORK
TITLE = Station B - Balk 1
      A     "Balk1";
      =     L 11.0;
      BLD   103;
      CALL  "SUB.Posit" (
           Station                  := "SIM.OB1".Balk_Station_B,
           BalkPostitie             := "SIM.OB1".Balk_1_boven,
           BalkNr                   := 1,
           BalkMerker               := L 11.0,
           Waarde                   := 128,
           ReturnStation            := #Return_StationB_Balk1,
           ActivatieStation         := #Activatie_StationB_Balk1);
      NOP   0;
NETWORK
TITLE = Station B - Balk 2
      A     "Blak2";
      =     L 11.0;
      BLD   103;
      CALL  "SUB.Posit" (
           Station                  := "SIM.OB1".Balk_Station_B,
           BalkPostitie             := "SIM.OB1".Balk_2_boven,
           BalkNr                   := 2,
           BalkMerker               := L 11.0,
           Waarde                   := 128,
           ReturnStation            := #Return_StationB_Balk2,
           ActivatieStation         := #Activatie_StationB_Balk2);
      NOP   0;
NETWORK
TITLE = Station B - Balk 3
      A     "Balk3";
      =     L 11.0;
      BLD   103;
      CALL  "SUB.Posit" (
           Station                  := "SIM.OB1".Balk_Station_B,
           BalkPostitie             := "SIM.OB1".Balk_3_boven,
           BalkNr                   := 3,
           BalkMerker               := L 11.0,
           Waarde                   := 128,
           ReturnStation            := #Return_StationB_Balk3,
           ActivatieStation         := #Activatie_StationB_Balk3);
      NOP   0;
NETWORK
TITLE = Station B - Balk 4
      A     "Balk4";
      =     L 11.0;
      BLD   103;
      CALL  "SUB.Posit" (
           Station                  := "SIM.OB1".Balk_Station_B,
           BalkPostitie             := "SIM.OB1".Balk_4_boven,
           BalkNr                   := 4,
           BalkMerker               := L 11.0,
           Waarde                   := 128,
           ReturnStation            := #Return_StationB_Balk4,
           ActivatieStation         := #Activatie_StationB_Balk4);
      NOP   0;
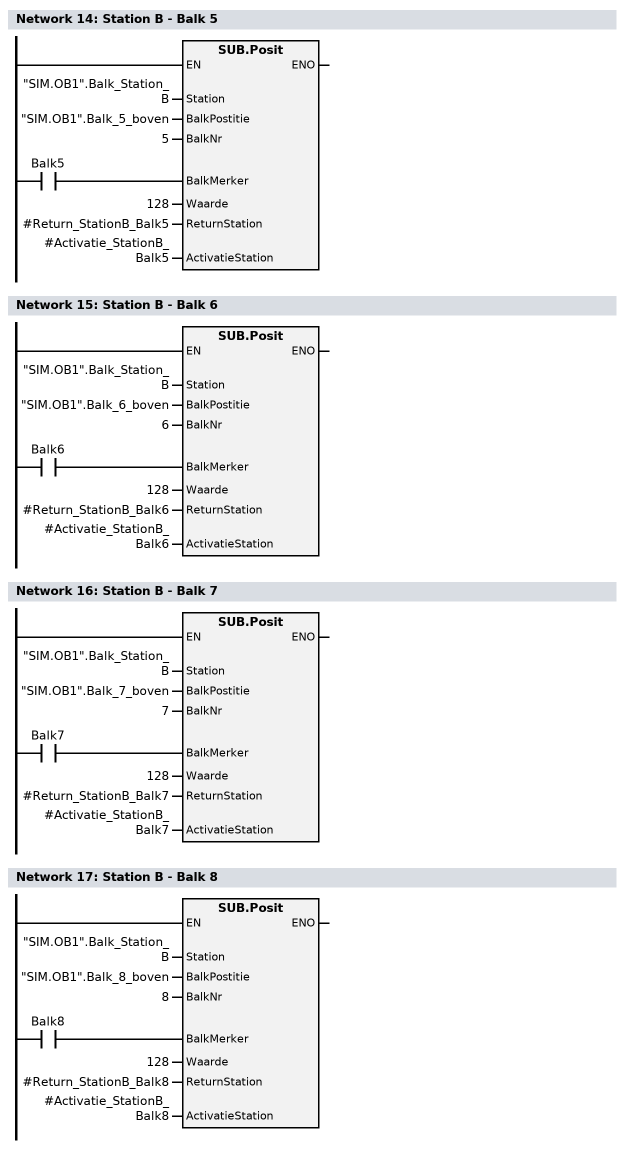
NETWORK
TITLE = Station B - Balk 5
      A     "Balk5";
      =     L 11.0;
      BLD   103;
      CALL  "SUB.Posit" (
           Station                  := "SIM.OB1".Balk_Station_B,
           BalkPostitie             := "SIM.OB1".Balk_5_boven,
           BalkNr                   := 5,
           BalkMerker               := L 11.0,
           Waarde                   := 128,
           ReturnStation            := #Return_StationB_Balk5,
           ActivatieStation         := #Activatie_StationB_Balk5);
      NOP   0;
NETWORK
TITLE = Station B - Balk 6
      A     "Balk6";
      =     L 11.0;
      BLD   103;
      CALL  "SUB.Posit" (
           Station                  := "SIM.OB1".Balk_Station_B,
           BalkPostitie             := "SIM.OB1".Balk_6_boven,
           BalkNr                   := 6,
           BalkMerker               := L 11.0,
           Waarde                   := 128,
           ReturnStation            := #Return_StationB_Balk6,
           ActivatieStation         := #Activatie_StationB_Balk6);
      NOP   0;
NETWORK
TITLE = Station B - Balk 7
      A     "Balk7";
      =     L 11.0;
      BLD   103;
      CALL  "SUB.Posit" (
           Station                  := "SIM.OB1".Balk_Station_B,
           BalkPostitie             := "SIM.OB1".Balk_7_boven,
           BalkNr                   := 7,
           BalkMerker               := L 11.0,
           Waarde                   := 128,
           ReturnStation            := #Return_StationB_Balk7,
           ActivatieStation         := #Activatie_StationB_Balk7);
      NOP   0;
NETWORK
TITLE = Station B - Balk 8
      A     "Balk8";
      =     L 11.0;
      BLD   103;
      CALL  "SUB.Posit" (
           Station                  := "SIM.OB1".Balk_Station_B,
           BalkPostitie             := "SIM.OB1".Balk_8_boven,
           BalkNr                   := 8,
           BalkMerker               := L 11.0,
           Waarde                   := 128,
           ReturnStation            := #Return_StationB_Balk8,
           ActivatieStation         := #Activatie_StationB_Balk8);
      NOP   0;
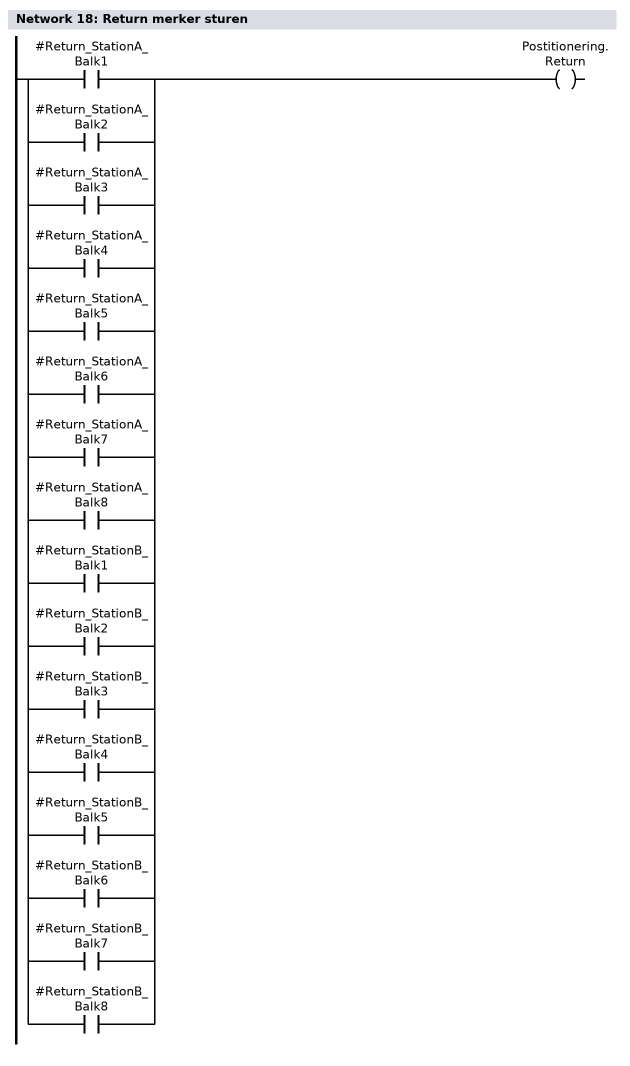
NETWORK
TITLE = Return merker sturen
      O     #Return_StationA_Balk1;
      O     #Return_StationA_Balk2;
      O     #Return_StationA_Balk3;
      O     #Return_StationA_Balk4;
      O     #Return_StationA_Balk5;
      O     #Return_StationA_Balk6;
      O     #Return_StationA_Balk7;
      O     #Return_StationA_Balk8;
      O     #Return_StationB_Balk1;
      O     #Return_StationB_Balk2;
      O     #Return_StationB_Balk3;
      O     #Return_StationB_Balk4;
      O     #Return_StationB_Balk5;
      O     #Return_StationB_Balk6;
      O     #Return_StationB_Balk7;
      O     #Return_StationB_Balk8;
      =     "Postitionering.Return";
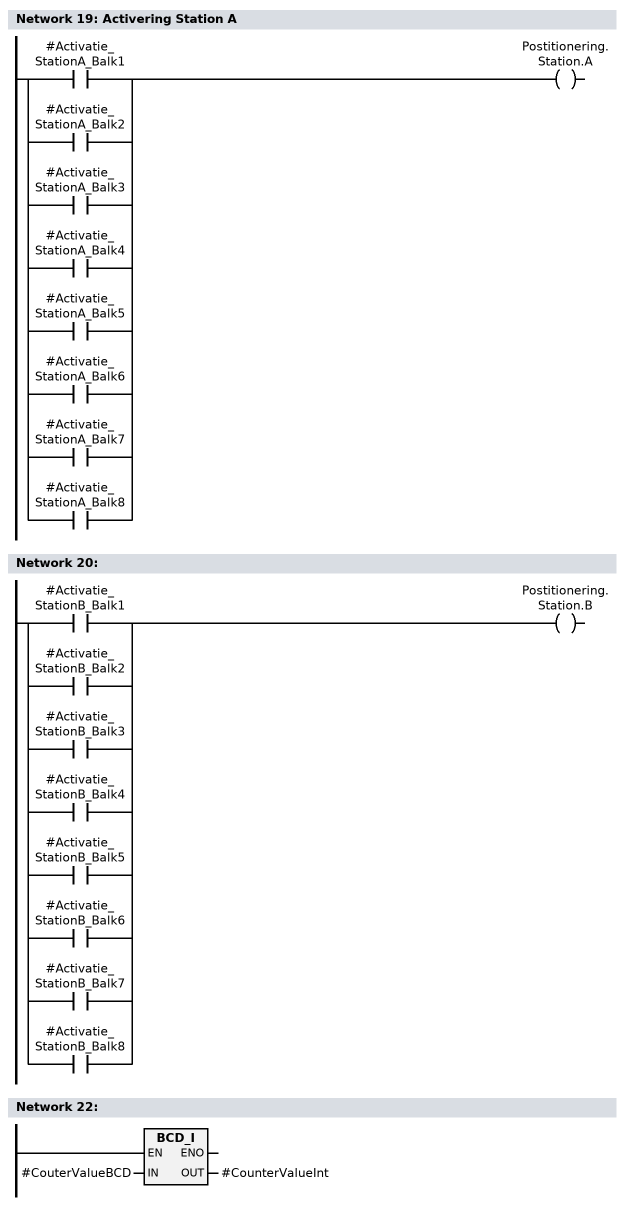
NETWORK
TITLE = Activering Station A
      O     #Activatie_StationA_Balk1;
      O     #Activatie_StationA_Balk2;
      O     #Activatie_StationA_Balk3;
      O     #Activatie_StationA_Balk4;
      O     #Activatie_StationA_Balk5;
      O     #Activatie_StationA_Balk6;
      O     #Activatie_StationA_Balk7;
      O     #Activatie_StationA_Balk8;
      =     "Postitionering.Station.A";
NETWORK
TITLE =
      O     #Activatie_StationB_Balk1;
      O     #Activatie_StationB_Balk2;
      O     #Activatie_StationB_Balk3;
      O     #Activatie_StationB_Balk4;
      O     #Activatie_StationB_Balk5;
      O     #Activatie_StationB_Balk6;
      O     #Activatie_StationB_Balk7;
      O     #Activatie_StationB_Balk8;
      =     "Postitionering.Station.B";
NETWORK
TITLE = Counter
      A(;
      O     "Postitionering.Station.A";
      O     "Postitionering.Station.B";
      O     "Postitionering.Return";
      );
      FP    #Positief;
      CU    "Positionering.counter";
      BLD   101;
      NOP   0;
      NOP   0;
      A     "Stap 2.0";
      R     "Positionering.counter";
      NOP   0;
      LC    "Positionering.counter";
      T     #CouterValueBCD;
      NOP   0;
NETWORK
TITLE =
      L     #CouterValueBCD;
      BTI;
      T     #CounterValueInt;
      NOP   0;
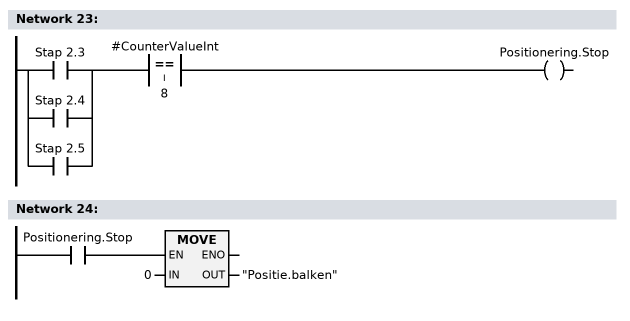
NETWORK
TITLE =
      A(;
      O     "Stap 2.3";
      O     "Stap 2.4";
      O     "Stap 2.5";
      );
      A(;
      L     #CounterValueInt;
      L     8;
      ==I;
      );
      =     "Positionering.Stop";
NETWORK
TITLE =
      A     "Positionering.Stop";
      JNB   _002;
      L     0;
      T     "Positie.balken";
_002: NOP   0;
END_FUNCTION

FUNCTION "Sub_routine" : VOID	// FC 14
VERSION : 0.1
VAR_INPUT
  voorwaarde : BOOL ;
END_VAR
VAR_IN_OUT
  huidige : BOOL ;
  volgende : BOOL ;
END_VAR
BEGIN
